TYPE HoursMinutesSeconds :
STRUCT
    positive : BOOL;
    
    hours : DINT;
    minutes : DINT;
    seconds : LREAL;
END_STRUCT
END_TYPE

(* stored: Version 1.1.0.1, ProductVersion 3.1.4018.5
   DUT HoursMinutesSeconds: Id {c29ce1e2-299a-43a5-a352-f76add1d4fa2} *)
